{attribute 'qualified_only'}
VAR_GLOBAL		
		fbLocalTime	:	FB_LocalSystemTime;
		iYear		:	UINT;
		iMonth		:	UINT;
		iDay		:	UINT;
		iHour		:	UINT;
		iMinute		:	UINT;
		iSecond		:	UINT;
END_VAR

(* stored: Version 1.1.0.1, ProductVersion 3.1.4024.12
   GVL GVL: Id {ff782142-a8f6-49f1-86c3-1589baad0be2} *)
